INTERFACE PUBLIC I_UnholdingCommands

METHOD PUBLIC Abort
END_METHOD

METHOD PUBLIC StateComplete
END_METHOD

METHOD PUBLIC Stop
END_METHOD

END_INTERFACE

(* stored: Version 1.1.0.1, ProductVersion 3.1.4026.6
   Itf I_UnholdingCommands: Id {2ed69181-4160-0c5d-1d9d-bb7c14caa326}
   Method Abort: Id {97561296-ba9d-404c-b71e-c6601771f0ea}
   Method StateComplete: Id {f7104005-8e40-4df9-a60a-9da8a56d408f}
   Method Stop: Id {85829acd-14cf-4d10-a737-445c3c38bcb5} *)
